FUNCTION alg_a_pusher2 : BOOL
VAR_INPUT
	state: STATE;
END_VAR

alg_a_pusher2 := state.dvar_M_inventory2_a_pusher2;

END_FUNCTION

(* stored: Version 1.1.0.1, ProductVersion 3.1.4022.18
   POU alg_a_pusher2: Id {3d5ddbc0-8a21-4c51-b2d1-9b2344c26c66}, SpecialFunc None *)
